PROGRAM PRG_MAIN
VAR
	fb_Blinking : ARRAY [0..1] OF FB_Blinking;
	fb_Exercice1: FB_Exercice1;
END_VAR


fb_Exercice1();

//fb_Blinking[0](Enable:=1 , PT_OFF:= , PT_ON:= , Output=>FIO_Output1[0]);
////fb_Blinking[1](Enable:=1 , PT_OFF:=T#1S, PT_ON:=T#3S, Output=>FIO_Output1[1]);

//IF FIO_I_Capteur THEN
//	FIO_O_Convoyeur := 1;
//ELSE
//	FIO_O_Convoyeur := 0;
//END_IF

END_PROGRAM

(* stored: Version 1.1.0.1, ProductVersion 3.1.4024.11
   POU PRG_MAIN: Id {11a895ac-5a06-4334-87ae-34581a64c27e}, SpecialFunc None *)
